(* Schneider Machine Expert - Basic project pump_pressure_control_TM221CE24T, file version 3.0.0.0 *)
(* ProjectInformations: Name=Pump Pressure Control with TM3AI4 *)

HARDWARE
  Cpu 0: TM221CE24T
  ModuleExtensionObject 0: TM3AI4/G
  EthernetConfiguration: NetworkName=M221, IpAllocationMode=ByDhcp, IpAddress=192.168.1.10, SubnetMask=255.255.255.0
  SerialLineConfiguration: Baud=Baud19200, Parity=ParityEven, DataBits=DataBits8, StopBits=StopBits1, PhysicalMedium=PhysicalMediumRs485, TransmissionMode=TransmissionModeModbusRtu, SlaveId=1, Addressing=SlaveAddressing
  MastTask: UsePeriodScanMode=false, PeriodScan=100
  FastTask: Period=255
  CpuBehavior: StartingMode=StartAsPreviousState, AutoSaveRamOnEeprom=true, WatchdogPeriod=250

SYMBOLS  (address, symbol, comment, settings)
  %M0       PUMP_RUN  "Pump running status"
  %M1       PRES_LOW  "Pressure below 5 bar"
  %M2       PRES_HIGH  "Pressure above 9.8 bar"
  %M3       AUTO_CMD  "Auto mode pump command"
  %M4       MAN_START  "Manual start command"
  %M5       AUTO_START  "Auto start command"
  %I0.0     PB_START
  %I0.1     PB_STOP
  %I0.2     ESTOP
  %I0.3     SS_AUTO
  %Q0.0     PUMP_OUT
  %Q0.1     LT_RUN
  %Q0.2     LT_AUTO
  %Q0.3     LT_PRES_HI
  %IW1.0    PRES_AIN  [Type=Type_4_20mA, Scope=Scope_Customized, Minimum=0, Maximum=10000]

POU Pump Pressure Control
  (* SectionNumber=0 *)

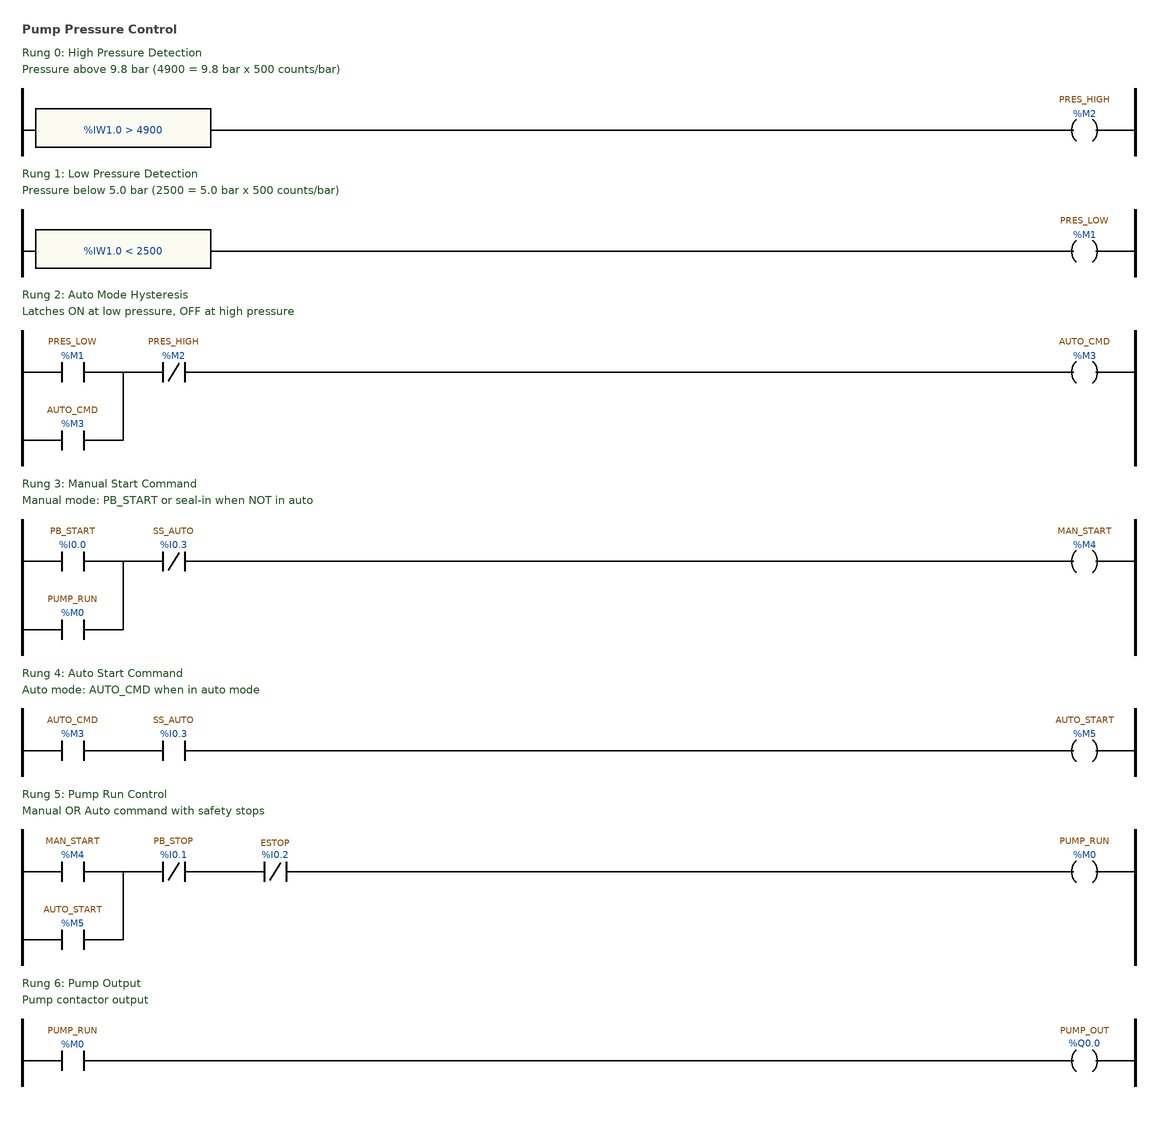

// Rung 0: High Pressure Detection
// Pressure above 9.8 bar (4900 = 9.8 bar x 500 counts/bar)
  LD [ %IW1.0 > 4900 ]    (* PRES_AIN *)
  ST %M2                  (* PRES_HIGH *)
  // as ST:
  //   PRES_HIGH := PRES_AIN > 4900;

// Rung 1: Low Pressure Detection
// Pressure below 5.0 bar (2500 = 5.0 bar x 500 counts/bar)
  LD [ %IW1.0 < 2500 ]    (* PRES_AIN *)
  ST %M1                  (* PRES_LOW *)
  // as ST:
  //   PRES_LOW := PRES_AIN < 2500;

// Rung 2: Auto Mode Hysteresis
// Latches ON at low pressure, OFF at high pressure
  LD %M1                  (* PRES_LOW *)
  OR %M3                  (* AUTO_CMD *)
  ANDN %M2                (* PRES_HIGH *)
  ST %M3                  (* AUTO_CMD *)
  // as ST:
  //   AUTO_CMD := (PRES_LOW OR AUTO_CMD) AND NOT PRES_HIGH;

// Rung 3: Manual Start Command
// Manual mode: PB_START or seal-in when NOT in auto
  LD %I0.0                (* PB_START *)
  OR %M0                  (* PUMP_RUN *)
  ANDN %I0.3              (* SS_AUTO *)
  ST %M4                  (* MAN_START *)
  // as ST:
  //   MAN_START := (PB_START OR PUMP_RUN) AND NOT SS_AUTO;

// Rung 4: Auto Start Command
// Auto mode: AUTO_CMD when in auto mode
  LD %M3                  (* AUTO_CMD *)
  AND %I0.3               (* SS_AUTO *)
  ST %M5                  (* AUTO_START *)
  // as ST:
  //   AUTO_START := AUTO_CMD AND SS_AUTO;

// Rung 5: Pump Run Control
// Manual OR Auto command with safety stops
  LD %M4                  (* MAN_START *)
  OR %M5                  (* AUTO_START *)
  ANDN %I0.1              (* PB_STOP *)
  ANDN %I0.2              (* ESTOP *)
  ST %M0                  (* PUMP_RUN *)
  // as ST:
  //   PUMP_RUN := (MAN_START OR AUTO_START) AND NOT PB_STOP AND NOT ESTOP;

// Rung 6: Pump Output
// Pump contactor output
  LD %M0                  (* PUMP_RUN *)
  ST %Q0.0                (* PUMP_OUT *)
  // as ST:
  //   PUMP_OUT := PUMP_RUN;

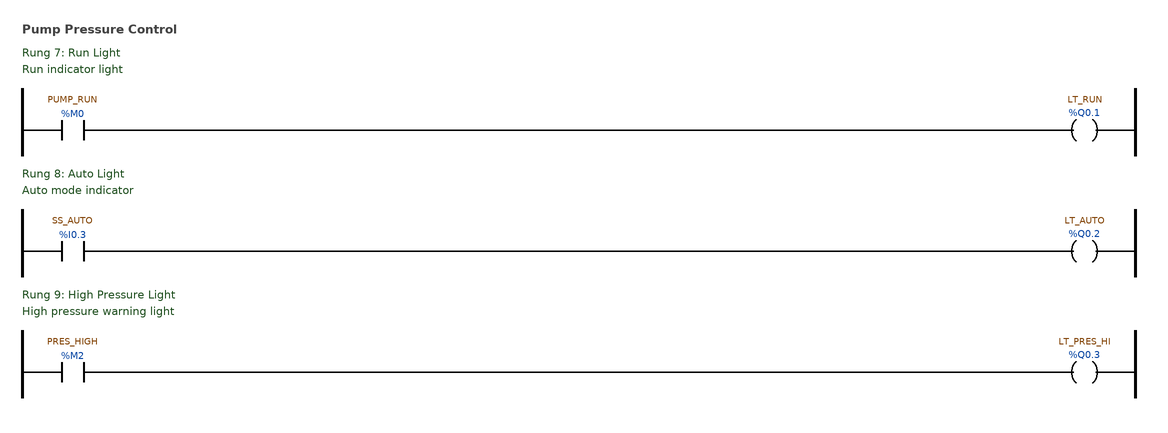

// Rung 7: Run Light
// Run indicator light
  LD %M0                  (* PUMP_RUN *)
  ST %Q0.1                (* LT_RUN *)
  // as ST:
  //   LT_RUN := PUMP_RUN;

// Rung 8: Auto Light
// Auto mode indicator
  LD %I0.3                (* SS_AUTO *)
  ST %Q0.2                (* LT_AUTO *)
  // as ST:
  //   LT_AUTO := SS_AUTO;

// Rung 9: High Pressure Light
// High pressure warning light
  LD %M2                  (* PRES_HIGH *)
  ST %Q0.3                (* LT_PRES_HI *)
  // as ST:
  //   LT_PRES_HI := PRES_HIGH;
